(* IEC 61131-3 sources: eCockpitGit/test_project/src/%F%00 Library/%F%JSON/%POU%FB_JSONWriter/%F%Write, 12 files *)

(* ---- %METH%writeBool.st ---- *)
//This adds a value data to the buffer
// |**Version**|**Author**| **Date** |**Changes**
// | 1         | NSN      | 22-06-20 | Creation
METHOD writeBool
VAR_INPUT
	value			:BOOL;				//Address of string for the filler text
END_VAR
VAR
	sTrue			:STRING(4) := 'true';
	sFalse			:STRING(5) := 'false';
END_VAR
(*%!%__DELIMITER__%!%*)
IF ready AND (afterKey OR_ELSE inArray OR_ELSE singleVal) THEN
	IF value THEN
		addString(pString:=ADR(sTrue));
	ELSE
		addString(pString:=ADR(sFalse));
	END_IF
	lastComma		:=		bufferPosition;
	addChar(char:=EASCII.Comma);
	//New line
	IF NOT(useSingleLine) AND NOT(treeSingleLine[treeLevel]) THEN
		addNewLine();
	END_IF
	afterKey		:=		FALSE;
	singleVal		:=		FALSE;
	emptyBlock		:=		FALSE;
END_IF

(* ---- %METH%writeDint.st ---- *)
//This adds a value data to the buffer
// |**Version**|**Author**| **Date** |**Changes**
// | 1         | NSN      | 22-06-20 | Creation
METHOD writeDint
VAR_INPUT
	value			:DINT;
END_VAR
VAR
	buffer			:STRING(11);
END_VAR
(*%!%__DELIMITER__%!%*)
IF ready AND (afterKey OR_ELSE inArray OR_ELSE singleVal) THEN
	buffer					:=		TO_STRING(value);
	addString(pString:=ADR(buffer));
	lastComma		:=		bufferPosition;
	addChar(char:=EASCII.Comma);
	IF NOT(useSingleLine) AND NOT(treeSingleLine[treeLevel]) THEN
		addNewLine();
	END_IF
	afterKey		:=		FALSE;
	singleVal		:=		FALSE;
	emptyBlock		:=		FALSE;
END_IF

(* ---- %METH%writeDword.st ---- *)
//This adds a value data to the buffer
// |**Version**|**Author**| **Date** |**Changes**
// | 1         | NSN      | 16-05-21 | Creation
METHOD writeDword
VAR_INPUT
	value			:DWORD;
END_VAR
VAR
	buffer			:STRING(10);
END_VAR
(*%!%__DELIMITER__%!%*)
IF ready AND (afterKey OR_ELSE inArray OR_ELSE singleVal) THEN
	buffer					:=		TO_STRING(value);
	addString(pString:=ADR(buffer));
	lastComma		:=		bufferPosition;
	addChar(char:=EASCII.Comma);
	IF NOT(useSingleLine) AND NOT(treeSingleLine[treeLevel]) THEN
		addNewLine();
	END_IF
	afterKey		:=		FALSE;
	singleVal		:=		FALSE;
	emptyBlock		:=		FALSE;
END_IF

(* ---- %METH%writeInt.st ---- *)
//This adds a value data to the buffer
// |**Version**|**Author**| **Date** |**Changes**
// | 1         | NSN      | 22-06-20 | Creation
METHOD writeInt
VAR_INPUT
	value			:INT;
END_VAR
VAR
	buffer			:STRING(6);
END_VAR
(*%!%__DELIMITER__%!%*)
IF ready AND (afterKey OR_ELSE inArray OR_ELSE singleVal) THEN
	buffer					:=		TO_STRING(value);
	addStringRaw(pString:=ADR(buffer));
	lastComma		:=		bufferPosition;
	addChar(char:=EASCII.Comma);
	IF NOT(useSingleLine) AND NOT(treeSingleLine[treeLevel]) THEN
		addNewLine();
	END_IF
	afterKey		:=		FALSE;
	singleVal		:=		FALSE;
	emptyBlock		:=		FALSE;
END_IF

(* ---- %METH%writeLint.st ---- *)
//This adds a value data to the buffer
// |**Version**|**Author**| **Date** |**Changes**
// | 1         | NSN      | 22-06-20 | Creation
METHOD writeLint
VAR_INPUT
	value			:LINT;
END_VAR
VAR
	buffer			:STRING(20);
END_VAR
(*%!%__DELIMITER__%!%*)
IF ready AND (afterKey OR_ELSE inArray OR_ELSE singleVal) THEN
	buffer					:=		TO_STRING(value);
	addString(pString:=ADR(buffer));
	lastComma		:=		bufferPosition;
	addChar(char:=EASCII.Comma);
	IF NOT(useSingleLine) AND NOT(treeSingleLine[treeLevel]) THEN
		addNewLine();
	END_IF
	afterKey		:=		FALSE;
	singleVal		:=		FALSE;
	emptyBlock		:=		FALSE;
END_IF

(* ---- %METH%writeLword.st ---- *)
//This adds a value data to the buffer
// |**Version**|**Author**| **Date** |**Changes**
// | 1         | NSN      | 16-05-21 | Creation
METHOD writeLword
VAR_INPUT
	value			:LWORD;
END_VAR
VAR
	buffer			:STRING(20);
END_VAR
(*%!%__DELIMITER__%!%*)
IF ready AND (afterKey OR_ELSE inArray OR_ELSE singleVal) THEN
	buffer					:=		TO_STRING(value);
	addString(pString:=ADR(buffer));
	lastComma		:=		bufferPosition;
	addChar(char:=EASCII.Comma);
	IF NOT(useSingleLine) AND NOT(treeSingleLine[treeLevel]) THEN
		addNewLine();
	END_IF
	afterKey		:=		FALSE;
	singleVal		:=		FALSE;
	emptyBlock		:=		FALSE;
END_IF

(* ---- %METH%writeNull.st ---- *)
//This adds a value data to the buffer
// |**Version**|**Author**| **Date** |**Changes**
// | 1         | NSN      | 22-06-20 | Creation
METHOD writeNull
VAR
	sNull			:STRING(4) := 'null';
END_VAR
(*%!%__DELIMITER__%!%*)
IF ready AND (afterKey OR_ELSE inArray OR_ELSE singleVal) THEN
	addString(pString:=ADR(sNull));
	lastComma		:=		bufferPosition;
	addChar(char:=EASCII.Comma);
	//New line
	IF NOT(useSingleLine) AND NOT(treeSingleLine[treeLevel]) THEN
		addNewLine();
	END_IF
	afterKey		:=		FALSE;
	singleVal		:=		FALSE;
	emptyBlock		:=		FALSE;
END_IF

(* ---- %METH%writeRaw.st ---- *)
//This adds a value data to the buffer
// |**Version**|**Author**| **Date** |**Changes**
// | 1         | NSN      | 22-06-20 | Creation
METHOD writeRaw
VAR_INPUT
	value			:POINTER TO EASCII;	//Address of string for the filler text
END_VAR
(*%!%__DELIMITER__%!%*)
IF ready AND (afterKey OR_ELSE inArray OR_ELSE singleVal) THEN
	addStringRaw(pString:=value);
	lastComma		:=		bufferPosition;
	addChar(char:=EASCII.Comma);
	IF NOT(useSingleLine) AND NOT(treeSingleLine[treeLevel]) THEN
		addNewLine();
	END_IF
	afterKey		:=		FALSE;
	singleVal		:=		FALSE;
	emptyBlock		:=		FALSE;
END_IF

(* ---- %METH%writeRawLen.st ---- *)
//This method writes a string of a fixed size to the buffer as raw data without qoutes and escape characters
//Should only be used for copying data
// |**Version**|**Author**| **Date** |**Changes**
// | 1         | NSN      | 13-10-21 | Creation
METHOD writeRawLen
VAR_INPUT
	value			:POINTER TO EASCII;	//Address of string for the filler text
	len				:DWORD;				//Amount of bytes to write
END_VAR
(*%!%__DELIMITER__%!%*)
IF ready AND (afterKey OR_ELSE inArray OR_ELSE singleVal) THEN
	addStringRawLen(pString:=value,len:=len);
	lastComma		:=		bufferPosition;
	addChar(char:=EASCII.Comma);
	IF NOT(useSingleLine) AND NOT(treeSingleLine[treeLevel]) THEN
		addNewLine();
	END_IF
	afterKey		:=		FALSE;
	singleVal		:=		FALSE;
	emptyBlock		:=		FALSE;
END_IF

(* ---- %METH%writeReal.st ---- *)
//This adds a value data to the buffer
// |**Version**|**Author**| **Date** |**Changes**
// | 1         | NSN      | 22-06-20 | Creation
METHOD writeReal
VAR_INPUT
	value			:REAL;
END_VAR
VAR
	buffer			:STRING(30);
	valuePoint		:POINTER TO DWORD := ADR(value);
END_VAR
(*%!%__DELIMITER__%!%*)
IF ready AND (afterKey OR_ELSE inArray OR_ELSE singleVal) THEN
	CASE valuePoint^ OF
		2139095040:	//Positive Infinity
			addChar(char:=EASCII.DoubleQoute);
			AddString(pString:=GTBigs.BInf);
			addChar(char:=EASCII.DoubleQoute);
		4286578688:	//Negative Infinity
			addChar(char:=EASCII.DoubleQoute);
			AddString(pString:=GTBigs.BminusInf);
			addChar(char:=EASCII.DoubleQoute);
		2143289344..2147483647,4290772992..4294967295:	//Not a Number
			addChar(char:=EASCII.DoubleQoute);
			AddString(pString:=GTBigs.BNaN);
			addChar(char:=EASCII.DoubleQoute);
	ELSE
		buffer					:=		TO_STRING(value);
		addString(pString:=ADR(buffer));
	END_CASE
	lastComma		:=		bufferPosition;
	addChar(char:=EASCII.Comma);
	IF NOT(useSingleLine) AND NOT(treeSingleLine[treeLevel]) THEN
		addNewLine();
	END_IF
	afterKey		:=		FALSE;
	singleVal		:=		FALSE;
	emptyBlock		:=		FALSE;
END_IF

(* ---- %METH%writeString.st ---- *)
//This adds a value data to the buffer
// |**Version**|**Author**| **Date** |**Changes**
// | 1         | NSN      | 22-06-20 | Creation
METHOD writeString
VAR_INPUT
	value			:POINTER TO EASCII;	//Address of string for the filler text
END_VAR
(*%!%__DELIMITER__%!%*)
IF ready AND (afterKey OR_ELSE inArray OR_ELSE singleVal) THEN
	addChar(char:=EASCII.DoubleQoute);
	AddString(pString:=value);
	addChar(char:=EASCII.DoubleQoute);
	lastComma		:=		bufferPosition;
	addChar(char:=EASCII.Comma);
	IF NOT(useSingleLine) AND NOT(treeSingleLine[treeLevel]) THEN
		addNewLine();
	END_IF
	afterKey		:=		FALSE;
	singleVal		:=		FALSE;
	emptyBlock		:=		FALSE;
END_IF

(* ---- %METH%writeWord.st ---- *)
//This adds a value data to the buffer
// |**Version**|**Author**| **Date** |**Changes**
// | 1         | NSN      | 16-05-21 | Creation
METHOD writeWord
VAR_INPUT
	value			:WORD;
END_VAR
VAR
	buffer			:STRING(5);
END_VAR
(*%!%__DELIMITER__%!%*)
IF ready AND (afterKey OR_ELSE inArray OR_ELSE singleVal) THEN
	buffer					:=		TO_STRING(value);
	addString(pString:=ADR(buffer));
	lastComma		:=		bufferPosition;
	addChar(char:=EASCII.Comma);
	IF NOT(useSingleLine) AND NOT(treeSingleLine[treeLevel]) THEN
		addNewLine();
	END_IF
	afterKey		:=		FALSE;
	singleVal		:=		FALSE;
	emptyBlock		:=		FALSE;
END_IF
